FUNCTION_BLOCK Real2_MatrixArray (* Basic FB with empty ECC *)
  (* Standard: 61499-2 *)
  (* Version 1.0, 2020-08-10, Candra Wardaya, UGM *)
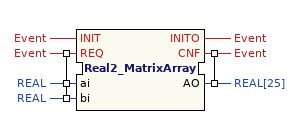
  EVENT_INPUT
    INIT; (* Initialization *)
    REQ WITH ai, bi; (* Normal Request of Execution *)
  END_EVENT
  EVENT_OUTPUT
    INITO; (* Initialization Output *)
    CNF WITH AO; (* Confirmation of Execution *)
  END_EVENT
  VAR_INPUT
    ai : REAL; (* Single Real Input *)
    bi : REAL; (* Single Real Input *)
  END_VAR
  VAR_OUTPUT
    AO : ARRAY [0..24] OF REAL; (* Array Input *)
  END_VAR
  VAR
    i : INT; (* Internal Variable *)
    val : REAL; (* Internal Variable *)
  END_VAR
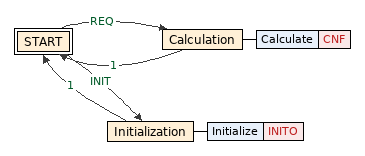
  EC_STATES
    START; (* Initial State *)
    Calculation : Calculate -> CNF;
    Initialization : Initialize -> INITO;
  END_STATES
  EC_TRANSITIONS
    Calculation TO START := 1;
    START TO Initialization := INIT;
    START TO Calculation := REQ;
    Initialization TO START := 1;
  END_TRANSITIONS
  ALGORITHM Calculate IN ST: (* New Algorithm *)
AO[0] := AO[0] + EXPT(ai,4);
AO[1] := AO[1] + (ai*ai)*(bi*bi);
AO[2] := AO[2] + (ai*ai)*(ai*bi);
AO[3] := AO[3] + (ai*ai)*ai;
AO[4] := AO[4] + (ai*ai)*bi;
AO[5] := AO[5] + (bi*bi)*(ai*ai); //[2][1]
AO[6] := AO[6] + (bi*bi)*(bi*bi);
AO[7] := AO[7] + (bi*bi)*(ai*bi);
AO[8] := AO[8] + (bi*bi)*(ai);
AO[9] := AO[9] + (bi*bi)*(bi);
AO[10] := AO[10] + (ai*bi)*(ai*ai); //[3][1]
AO[11] := AO[11] + (ai*bi)*(bi*bi);
AO[12] := AO[12] + (ai*bi)*(ai*bi);
AO[13] := AO[13] + (ai*bi)*(ai);
AO[14] := AO[14] + (ai*bi)*(bi);
AO[15] := AO[15] + (ai)*(ai*ai);//[4][1]
AO[16] := AO[16] + (ai)*(bi*bi);
AO[17] := AO[17] + (ai)*(ai*bi);
AO[18] := AO[18] + (ai)*(ai);
AO[19] := AO[19] + (ai)*(bi);
AO[20] := AO[20] + (bi)*(ai*ai); //[5][1]
AO[21] := AO[21] + (bi)*(bi*bi);
AO[22] := AO[22] + (bi)*(ai*bi);
AO[23] := AO[23] + (bi)*(ai);
AO[24] := AO[24] + (bi)*(bi);
  END_ALGORITHM
  ALGORITHM Initialize IN ST: (* New Algorithm *)

  END_ALGORITHM
END_FUNCTION_BLOCK
